FUNCTION F_FormatString10 : T_MaxString
VAR_INPUT
	Format	: T_MaxString;
	arg1	: T_Arg;
	arg2	: T_Arg;
	arg3	: T_Arg;
	arg4	: T_Arg;
	arg5	: T_Arg;
	arg6	: T_Arg;
	arg7	: T_Arg;
	arg8	: T_Arg;
	arg9	: T_Arg;
	arg10	: T_Arg;
END_VAR
VAR
    FB_FormatString1 : FB_FormatString;
END_VAR

FB_FormatString1(
	sFormat:= Format, 
	arg1:= arg1, 
	arg2:= arg2, 
	arg3:= arg3, 
	arg4:= arg4, 
	arg5:= arg5, 
	arg6:= arg6, 
	arg7:= arg7, 
	arg8:= arg8, 
	arg9:= arg9, 
	arg10:= arg10, 
	bError=> , 
	nErrId=> , 
	sOut=> F_FormatString10);

END_FUNCTION

(* stored: Version 1.1.0.1, ProductVersion 3.1.4024.3
   POU F_FormatString10: Id {16584a81-b5c5-0f45-18a0-ad7a781fd9ec}, SpecialFunc None *)
